// TwinCAT 3 PLC project plc
// ProgramVersion: 3.1.4026.24
// libraries:
//   Tc2_Standard, * (Beckhoff Automation GmbH)
//   Tc2_System, * (Beckhoff Automation GmbH)
// project tree:
//   DUTs/ ST_Datos.TcDUT
//   / PlcTask.TcTTO
//   POUs/ MAIN.TcPOU
// real-time tasks:
//   TASK PlcTask: cycle T#10ms, priority 20, ADS port 350

CONFIGURATION plc
    RESOURCE PLC ON TwinCAT3
        TASK PlcTask(INTERVAL := T#10ms, PRIORITY := 20);
        PROGRAM MAIN WITH PlcTask : MAIN;
    END_RESOURCE
END_CONFIGURATION

// ---- DUTs/ST_Datos.TcDUT
TYPE ST_Datos :
STRUCT
	nNumber		: INT;
	bBool		: BOOL;
	rValue1		: REAL;
END_STRUCT
END_TYPE

// ---- POUs/MAIN.TcPOU
PROGRAM MAIN
VAR
	bInit		: BOOL := TRUE;
	i			: INT;
	aDatos		: ARRAY[1..100] OF ST_Datos;
END_VAR

IF bInit THEN
	FOR i:=1 TO 100 DO
		aDatos[i].rValue1 := i*10.0;
		aDatos[i].nNumber := i;
	END_FOR
	bInit := FALSE;
END_IF

END_PROGRAM
